TYPE STATE:
    STRUCT
        curTime: LREAL;
        dvar_M_aut_y: DINT;
    END_STRUCT;
END_TYPE
